(* PLC project My_Firt_Project, Desconhecido Sem nome 1 *)
(* stored: creationDateTime 2022-02-03T12:16:02, modificationDateTime 2022-02-03T12:37:59 *)

PROGRAM My_First_Program
  VAR
    PB1 AT %IX100.0 : BOOL;
    PB2 AT %IX100.1 : BOOL;
    LED AT %QX100.0 : BOOL;
  END_VAR

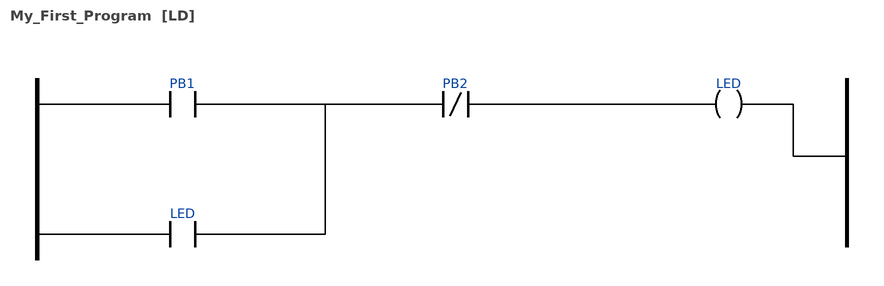
(* LD diagram, written out as Structured Text *)
LED := (PB1 OR LED) AND NOT PB2;
END_PROGRAM

CONFIGURATION Config0
  RESOURCE Res0 ON PLC
    TASK task0(INTERVAL := T#20ms, PRIORITY := 0);
    PROGRAM instance0 WITH task0 : My_First_Program;
  END_RESOURCE
END_CONFIGURATION
